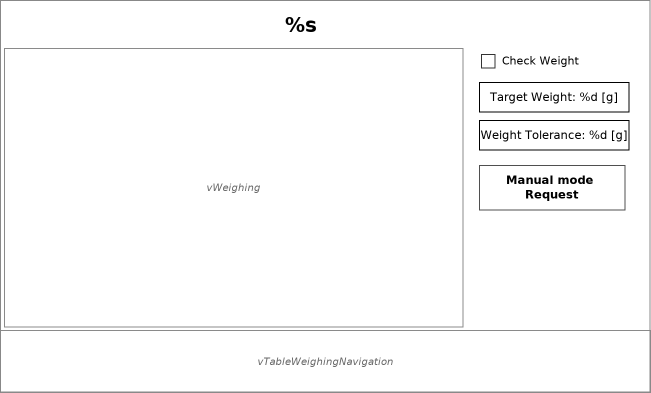
VISUALIZATION vTableWeighingWeight  // 651x393
VAR_IN_OUT
	fbStation:FB_WeighingStation;
	fbTableControl: FB_TableControl;
END_VAR
    Rectangle (0,0 650x392)
    Rectangle (226,10 150x30), "%s", text variable: fbStation.sStationName
    Rectangle (479,120 150x30), "Weight Tolerance: %d [g]", text variable: fbStation.stSettings.stWeighingBottleParams.rWeightTolerance
        OnMouseClick: write the text variable via Default, min 0, format %d
    Rectangle (479,82 150x30), "Target Weight: %d [g]", text variable: fbStation.stSettings.stWeighingBottleParams.rTargetWeight
        OnMouseClick: write the text variable via Default, min 0, format %d
    Frame (0,330 651x63)
        shows vTableWeighingNavigation(fbTableControl := fbTableControl)
    Checkbox (479,46 150x30), "Check Weight", variable: fbStation.stSettings.bWeightCheck
    Rectangle (479,165 146x45), "Manual mode Request", colour toggle: fbStation.bManualModeRequest
        toggle fbStation.bManualModeRequest
    Frame (4,48 459x279)
        shows vWeighing(iNameIndex := 4, fbWeighing := fbStation.fbWeighing)
END_VISUALIZATION

(* stored: Version 1.1.0.1, ProductVersion 3.1.4024.15
   Visu vTableWeighingWeight: Id {1e5ba465-b682-4cdd-b2f8-82aa8ecf87c2} *)
